// TIA Portal project "PLCtilWinSocket1" (V13)

(* hardware
DEVICE "S7-1200 station_1"  S7-1200 Station
   slot 0: "Rack_0"  Rack  V1.0
   slot 1: "PLC_1"  CPU 1214C DC/DC/DC  6ES7 214-1AG40-0XB0  V4.1
   slot 3: "AQ 1x12BIT_1"  6ES7 232-4HA30-0XB0  V1.0
*)

// ===== PLC "PLC_1"  CPU 1214C DC/DC/DC =====

VAR_GLOBAL   // PLC tag table "Default tag table"
   "EnableForbindelse" AT %I0.0 : Bool;
   "EnableSend" AT %I0.1 : Bool;
   "EnableModtag" AT %I0.2 : Bool;
   "DisableForbindelse" AT %I0.3 : Bool;
END_VAR

DATA_BLOCK "Data"   // DB4
{ S7_Optimized_Access := 'FALSE' }
VERSION : 0.1
   VAR
      ModtagData : Word;
      SendData : Array[0..3] of Char;
      SendData1 : Char;
      StringData : String;
      IntegerData : UInt;
      Format : Word;
      countChars : UInt;
   END_VAR
BEGIN
END_DATA_BLOCK

// folder: System blocks/Program resources

DATA_BLOCK "PLC_1_Connection_DB"   // DB2
{ S7_Optimized_Access := 'FALSE' }
AUTHOR : SIMATIC
FAMILY : MC7Plus
NAME : TC_IP_v4
VERSION : 1.0
// stored: InstanceOfName ?
"?"
BEGIN
END_DATA_BLOCK

// folder: (top level)

FUNCTION "OpretForbindelse" : Void   // FC1, LAD
{ S7_Optimized_Access := 'FALSE' }
VERSION : 0.1
BEGIN

REGION Network 1
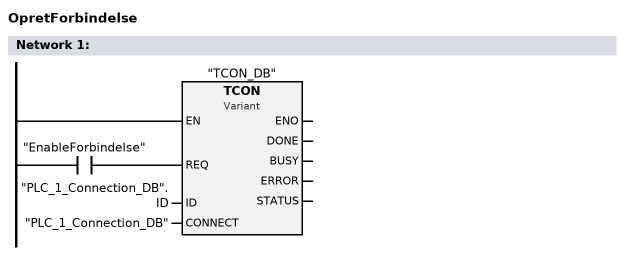
   "TCON_DB"(REQ := "EnableForbindelse", ID := "PLC_1_Connection_DB".ID, CONNECT := "PLC_1_Connection_DB");   // TCON
END_REGION
END_FUNCTION

FUNCTION "Modtag" : Void   // FC2, LAD
{ S7_Optimized_Access := 'FALSE' }
VERSION : 0.1
BEGIN

REGION Network 1: Modtag data
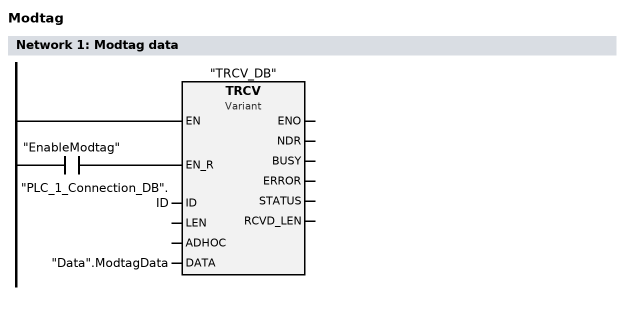
   "TRCV_DB"(EN_R := "EnableModtag", ID := "PLC_1_Connection_DB".ID, DATA := "Data".ModtagData);   // TRCV
END_REGION
END_FUNCTION

FUNCTION "Send" : Void   // FC3, LAD
{ S7_Optimized_Access := 'FALSE' }
VERSION : 0.1
BEGIN

REGION Network 1
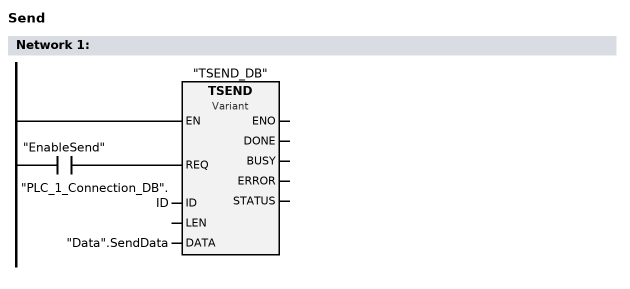
   "TSEND_DB"(REQ := "EnableSend", ID := "PLC_1_Connection_DB".ID, DATA := "Data".SendData);   // TSEND
END_REGION
END_FUNCTION

FUNCTION "AfslutForbindelse" : Void   // FC4, LAD
{ S7_Optimized_Access := 'FALSE' }
VERSION : 0.1
BEGIN

REGION Network 1
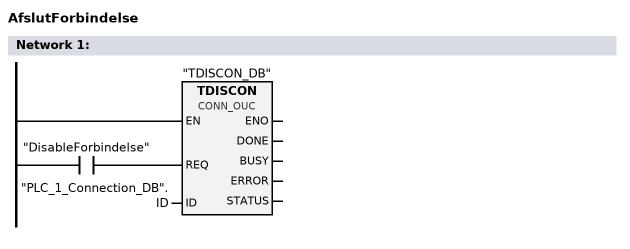
   "TDISCON_DB"(REQ := "DisableForbindelse", ID := "PLC_1_Connection_DB".ID);   // TDISCON
END_REGION
END_FUNCTION

ORGANIZATION_BLOCK "Main"   // OB1, LAD, ProgramCycle
TITLE = "Main Program Sweep (Cycle)"
{ S7_Optimized_Access := 'FALSE' }
VERSION : 0.1
BEGIN

REGION Network 1: Opret forbindelse
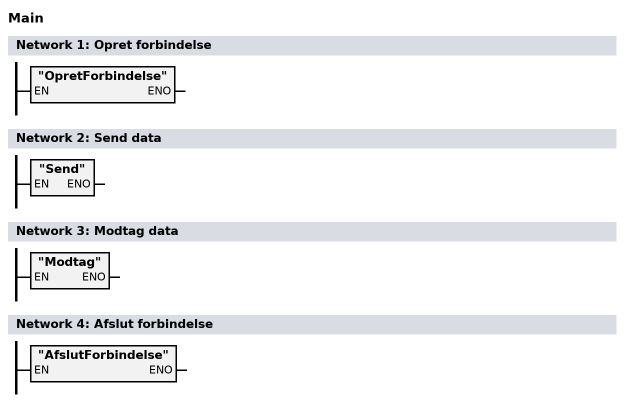
   RUNG wire#powerrail
      "OpretForbindelse"()
   END_RUNG
   // the same network as SCL:
   "OpretForbindelse"();
END_REGION

REGION Network 2: Send data
   RUNG wire#powerrail
      "Send"()
   END_RUNG
   // the same network as SCL:
   "Send"();
END_REGION

REGION Network 3: Modtag data
   RUNG wire#powerrail
      "Modtag"()
   END_RUNG
   // the same network as SCL:
   "Modtag"();
END_REGION

REGION Network 4: Afslut forbindelse
   RUNG wire#powerrail
      "AfslutForbindelse"()
   END_RUNG
   // the same network as SCL:
   "AfslutForbindelse"();
END_REGION

REGION Network 5: Kommunikationsstyring
END_REGION
END_ORGANIZATION_BLOCK